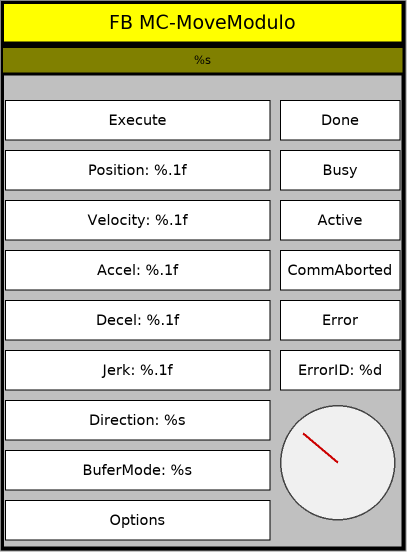
VISUALIZATION MC_MoveModulo2  // 407x552
VAR_INPUT
	{attribute 'parameterstringof' := 'm_Input_FB_Modulo'}
	m_Input_FB_Modulo_Str : STRING;
END_VAR
VAR_IN_OUT
	m_Input_FB_Modulo : None;
END_VAR
    Rectangle (0,0 405x550)
    Rectangle (5,100 265x40), "Execute", colour toggle: (m_Input_FB_Modulo.Execute) <> 0
        toggle m_Input_FB_Modulo.Execute
    Rectangle (5,150 265x40), "Position: %.1f", text variable: m_Input_FB_Modulo.Position
        OnMouseDown: write the text variable via Edit
    Rectangle (5,200 265x40), "Velocity: %.1f", text variable: m_Input_FB_Modulo.Velocity
        OnMouseDown: write the text variable via Edit
    Rectangle (5,250 265x40), "Accel: %.1f", text variable: m_Input_FB_Modulo.Acceleration
        OnMouseDown: write the text variable via Edit
    Rectangle (5,300 265x40), "Decel: %.1f", text variable: m_Input_FB_Modulo.Deceleration
        OnMouseDown: write the text variable via Edit
    Rectangle (5,350 265x40), "Jerk: %.1f", text variable: m_Input_FB_Modulo.Jerk
    Rectangle (5,400 265x40), "Direction: %s", text variable: m_Input_FB_Modulo.Direction
        OnMouseDown: write the text variable via VisuDialogs.Numpad
    Rectangle (5,450 265x40), "BuferMode: %s", tooltip "TYPE MC_BufferMode : ( MC_Aborting := 16#00, MC_Buffered := 16#01, MC_BlendingLow := 16#12, MC_BlendingPrevious := 16#13, MC_BlendingNext := 16#14, MC_BlendingHigh := 16#15 ); END_TYPE", text variable: m_Input_FB_Modulo.BufferMode
    Rectangle (5,500 265x40), "Options"
    Rectangle (280,100 120x40), "Done", colour toggle: (m_Input_FB_Modulo.Done) <> 0
    Rectangle (280,150 120x40), "Busy", colour toggle: (m_Input_FB_Modulo.Busy) <> 0
    Rectangle (280,200 120x40), "Active", colour toggle: (m_Input_FB_Modulo.Active) <> 0
    Rectangle (280,250 120x40), "CommAborted", colour toggle: (m_Input_FB_Modulo.CommandAborted) <> 0
    Rectangle (280,300 120x40), "Error", colour toggle: (m_Input_FB_Modulo.Error) <> 0
    Rectangle (280,350 120x40), "ErrorID: %d", text variable: m_Input_FB_Modulo.ErrorID
    Rectangle (0,0 405x45), "FB MC-MoveModulo"
    Meter (280,405 115x115), value: $FB_Modulo$.Axis.NcToPlc.ModuloActPos, scale format: %.f, scale 0..270
    Rectangle (0,45 405x30), "%s", text variable: m_Input_FB_Modulo_Str
END_VISUALIZATION

(* stored: Version 1.1.0.1, ProductVersion 3.1.4024.11
   Visu MC_MoveModulo2: Id {e928230e-d7ab-4858-be9f-9d5d7d2cdb3a} *)
